Fanuc KAREL source: SET_TRNS_TPE.kl

PROGRAM T
%NOLOCKGROUP
VAR
 v0 : INTEGER
 v1 : INTEGER
 v2 : POSITION
 v3 : INTEGER
BEGIN
 SET_TRNS_TPE(v0, v1, v2, v3)
END T
